FUNCTION_BLOCK PublishEventHTTP (* Publish event using HTTP *)
  (* Standard: 61499-2; Description: Copyright (c) 2019 fortiss GmbH This program and the accompanying materials are made available under the terms of the Eclipse Public License 2.0 which is available at https://www.eclipse.org/legal/epl-2.0/ SPDX-License-Identifier: EPL-2.0 *)
  (* Version 1.0, 2019-09-17, Cabral, fortiss GmbH *)
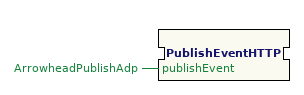
  SOCKETS
    publishEvent : ArrowheadPublishAdp; (* Publish Event adapter *)
  END_SOCKETS
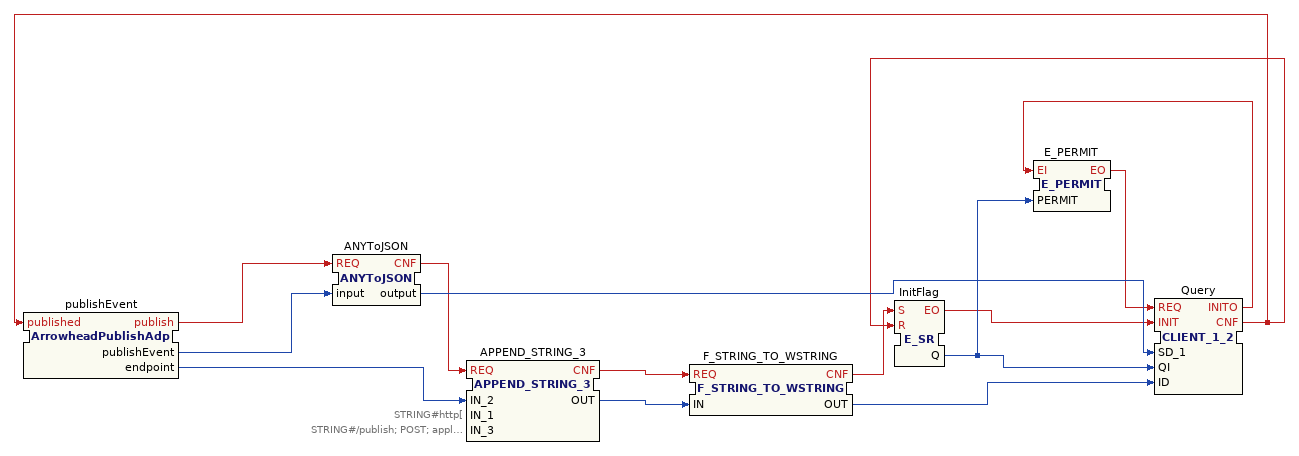
  FBS
    ANYToJSON : ANYToJSON;
    InitFlag : E_SR;
    APPEND_STRING_3 : APPEND_STRING_3(IN_1 := STRING#http[, IN_3 := STRING#/publish; POST; application/json]);
    F_STRING_TO_WSTRING : F_STRING_TO_WSTRING;
    Query : CLIENT_1_2;
    E_PERMIT : E_PERMIT;
  END_FBS
  EVENT_CONNECTIONS
    E_PERMIT.EO TO Query.REQ;
    APPEND_STRING_3.CNF TO F_STRING_TO_WSTRING.REQ;
    InitFlag.EO TO Query.INIT;
    ANYToJSON.CNF TO APPEND_STRING_3.REQ;
    F_STRING_TO_WSTRING.CNF TO InitFlag.S;
    Query.INITO TO E_PERMIT.EI;
    Query.CNF TO InitFlag.R;
    publishEvent.publish TO ANYToJSON.REQ;
    Query.CNF TO publishEvent.published;
  END_CONNECTIONS
  DATA_CONNECTIONS
    ANYToJSON.output TO Query.SD_1;
    InitFlag.Q TO Query.QI;
    APPEND_STRING_3.OUT TO F_STRING_TO_WSTRING.IN;
    F_STRING_TO_WSTRING.OUT TO Query.ID;
    InitFlag.Q TO E_PERMIT.PERMIT;
    publishEvent.publishEvent TO ANYToJSON.input;
    publishEvent.endpoint TO APPEND_STRING_3.IN_2;
  END_CONNECTIONS
END_FUNCTION_BLOCK
